// TwinCAT 3 PLC project TypesTest
// ProgramVersion: 3.1.4024.0
// libraries:
//   Tc3_Module, * (Beckhoff Automation GmbH)
//   TcUnit, * (www.tcunit.org)
//   Types, * (TomasRompotl)
// project tree:
//   Binding/ BindTest.TcPOU, BoolBindingReadOnlyTest.TcPOU, NotBindTest.TcPOU (not stored)
//   / PlcTask.TcTTO (not stored), PRG_Test.TcPOU (not stored)
//   Reflection/ ReflectionTest.TcPOU
//   Values/BooleanExpression/ BooleanExpressionFunctionsTest.TcPOU (not stored), BooleanExpressionTest.TcPOU (not stored)
//   Values/ BoolValuesTest.TcPOU (not stored)
// real-time tasks:
//   TASK TypesTestTask: cycle T#1ms, priority 20, ADS port 350
//   TASK StringsTestTask: cycle T#1ms, priority 21, ADS port 351
//   TASK DataTestTask: cycle T#1ms, priority 22, ADS port 352
//   TASK MathTestTask: cycle T#1ms, priority 23, ADS port 353
//   TASK TimesTestTask: cycle T#1ms, priority 24, ADS port 354

// ---- Binding/BindTest.TcPOU
FUNCTION_BLOCK BindTest EXTENDS TcUnit.FB_TestSuite
VAR
END_VAR

BindAndTestBinding();

METHOD BindAndTestBinding : BOOL
VAR
	expected : BOOL;
	actual : BOOL;
	
	variable : BOOL;
	binding : BoolValue;
	disposable : Disposable;
END_VAR
TcUnit.TEST('Bind and test binding');

binding := Bind(variable);

expected := TRUE;
actual := binding <> 0;

AssertEquals(
	Expected := expected,
	Actual := actual,
	Message := 'Bind should return interface to created Binding');
	
variable := TRUE;

expected := TRUE;
actual := binding.Value;

AssertEquals(
	Expected := expected,
	Actual := actual,
	Message := 'Binding should return value of binded variable');
	
__QUERYINTERFACE(binding, disposable);
disposable.Dispose();

TEST_FINISHED();
END_METHOD

END_FUNCTION_BLOCK

// ---- Binding/BoolBindingReadOnlyTest.TcPOU
FUNCTION_BLOCK BoolBindingReadOnlyTest EXTENDS TcUnit.FB_TestSuite
VAR
END_VAR

CheckIsBinded();
BindingReturnsSameValue();
NegatedBindingReturnsNegatedValue();

METHOD BindingReturnsSameValue : BOOL
VAR
	expected : BOOL;
	actual : BOOL;
	
	binding : BoolBindingReadOnly;
	variable : BOOL;
END_VAR
TcUnit.TEST('Binding returns same value');

binding.Bind(variable);

expected := FALSE;
actual := binding.Value;

AssertEquals(
	Expected := expected,
	Actual := actual,
	Message := 'Value should return FALSE if binded variable is FALSE');
	
variable := TRUE;

expected := TRUE;
actual := binding.Value;

AssertEquals(
	Expected := expected,
	Actual := actual,
	Message := 'Value should return TRUE if binded variable is TRUE');

TEST_FINISHED();
END_METHOD

METHOD CheckIsBinded : BOOL
VAR
	expected : BOOL;
	actual : BOOL;
	
	binding : BoolBindingReadOnly;
	variable : BOOL;
END_VAR
TcUnit.TEST('Check binded');

expected := FALSE;
actual := binding.IsBinded;

AssertEquals(
	Expected := expected,
	Actual := actual,
	Message := 'IsBinded should be FALSE before binding');

binding.Bind(variable);

expected := TRUE;
actual := binding.IsBinded;

AssertEquals(
	Expected := expected,
	Actual := actual,
	Message := 'IsBinded should be TRUE after successful Bind()');

TEST_FINISHED();
END_METHOD

METHOD NegatedBindingReturnsNegatedValue : BOOL
VAR
	expected : BOOL;
	actual : BOOL;
	
	binding : BoolBindingReadOnly;
	variable : BOOL;
END_VAR
TcUnit.TEST('Negated binding returns negated value');

binding.Bind(variable);
binding.Negate := TRUE;

expected := TRUE;
actual := binding.Value;

AssertEquals(
	Expected := expected,
	Actual := actual,
	Message := 'Value should return TRUE if binded variable is FALSE');
	
variable := TRUE;

expected := FALSE;
actual := binding.Value;

AssertEquals(
	Expected := expected,
	Actual := actual,
	Message := 'Value should return FALSE if binded variable is TRUE');

TEST_FINISHED();
END_METHOD

END_FUNCTION_BLOCK

// ---- Reflection/ReflectionTest.TcPOU
FUNCTION_BLOCK ReflectionTest EXTENDS TcUnit.FB_TestSuite
VAR
	reflection : Reflection(THIS, SIZEOF(THIS^));
END_VAR

GetAllData();

METHOD GetAllData : BOOL
VAR
END_VAR
TcUnit.TEST('Get all data');

AssertEquals_STRING(
	Actual := reflection.InstanceName,
	Expected := 'FrameworkMonorepoTests.TypesTest.PRG_Test.reflectionTest',
	Message := 'InstanceName was not obtained correctly');

AssertEquals_STRING(
	Actual := reflection.SolutionName,
	Expected := 'FrameworkMonorepoTests',
	Message := 'SolutionName was not obtained correctly');

AssertEquals_STRING(
	Actual := reflection.ProjectName,
	Expected := 'TypesTest',
	Message := 'ProjectName was not obtained correctly');

AssertEquals_STRING(
	Actual := reflection.ParentName,
	Expected := 'PRG_Test',
	Message := 'ParentName was not obtained correctly');

AssertEquals_STRING(
	Actual := reflection.Name,
	Expected := 'reflectionTest',
	Message := 'Name was not obtained correctly');

AssertEquals_STRING(
	Actual := reflection.ObjectPath,
	Expected := 'PRG_Test.reflectionTest',
	Message := 'ObjectPath was not obtained correctly');

AssertEquals_STRING(
	Actual := reflection.TypeName,
	Expected := 'ReflectionTest',
	Message := 'TypeName was not obtained correctly');

TEST_FINISHED();
END_METHOD

END_FUNCTION_BLOCK
